// Mitsubishi GX Works2 project: 0319_인터로크3   PLC: Q03UDV

PROGRAM MAIN
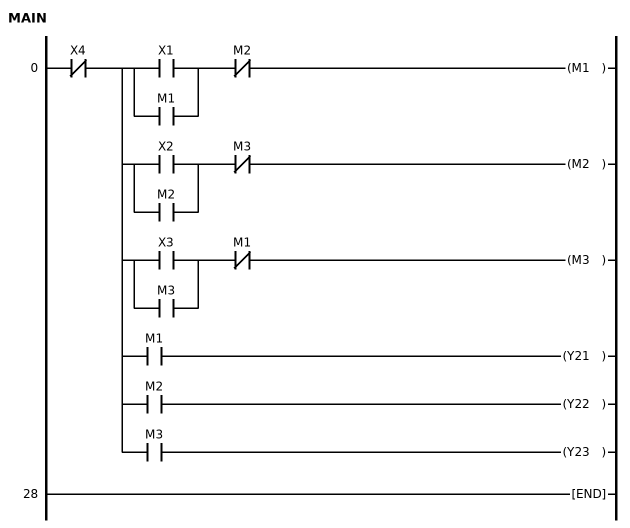
0     LDI     X4
      MPS
      LD      X1
      OR      M1
      ANB
      ANI     M2
      OUT     M1
      MRD
      LD      X2
      OR      M2
      ANB
      ANI     M3
      OUT     M2
      MRD
      LD      X3
      OR      M3
      ANB
      ANI     M1
      OUT     M3
      MRD
      AND     M1
      OUT     Y21
      MRD
      AND     M2
      OUT     Y22
      MPP
      AND     M3
      OUT     Y23
28    END
END_PROGRAM
